INTERFACE I_STOP_GATE EXTENDS I_GENERAL_OBJECT

METHOD M_Close
VAR_INPUT
END_VAR
END_METHOD

METHOD M_Open
VAR_INPUT
END_VAR
END_METHOD

METHOD M_Seperate
VAR_INPUT
	iCntCarrier: INT;
END_VAR
END_METHOD

PROPERTY P_CarrierByStopGate : BOOL
GET
END_GET
END_PROPERTY

PROPERTY P_Congestion : BOOL
GET
END_GET
END_PROPERTY

END_INTERFACE

(* stored: Version 1.1.0.1, ProductVersion 3.1.4024.12
   Itf I_STOP_GATE: Id {d2545a88-d905-4266-b7ff-b4ed84ac9176}
   Method M_Close: Id {9010d98f-dc8a-4065-83b3-965b8a7191e0}
   Method M_Open: Id {fc3288e5-9699-4262-a557-3e9d4cda5436}
   Method M_Seperate: Id {959ae008-8bb0-4b17-ad33-8b9bbea65977}
   Property P_CarrierByStopGate: Id {5d520a10-f556-4676-96fc-f08b795439bc}
   Get Get: Id {c92f1a23-7dc5-426a-87ea-d9fb607700ee}
   Property P_Congestion: Id {e0aa719d-a570-4c33-a415-eb090448b3c6}
   Get Get: Id {22a5db1c-d2e3-4446-9e87-26f677ae3798} *)
